// Mitsubishi GX Works2 project: SPMDanNhanV1   PLC: FX3G

// global labels: Global1
VAR_GLOBAL
  SIGNAL_JAR AT X000 : BOOL;
  SIGNAL_LABEL AT X001 : BOOL;
  EMERG AT X007 : BOOL;
  LABEL_PLS AT Y000 : BOOL;
  LABEL_DIR AT Y003 : BOOL;
  PushManLabel_F AT M200 : BOOL;
  PushManLabel_R AT M201 : BOOL;
  PushManGird_F AT M202 : BOOL;
  PushManGird_R AT M203 : BOOL;
  PushManRulo_F AT M204 : BOOL;
  PushManRulo_R AT M205 : BOOL;
  ModeAuto AT M206 : BOOL;
  Alarm AT M207 : BOOL;
  Operation AT M208 : BOOL;
  Speed_Label AT D200 : DINT;
  Length_Label AT D202 : DINT;
  Speed_Stamp AT D204 : DINT;
  Length_Stamp AT D206 : DINT;
  Round_Gird AT D208 : DINT;
  Round_Rulo AT D210 : DINT;
  Reset AT M209 : BOOL;
  Restore AT M210 : BOOL;
  FullStep_Label AT D212 : DINT;
  CommandLabel1 : BOOL;
  CommandLabel2 : BOOL;
  LABEL_ENB AT Y004 : BOOL;
  GIRD_PLS AT Y001 : BOOL;
  RULO_PLS AT Y002 : BOOL;
  RULO_ENB AT Y006 : BOOL;
  GIRD_ENB AT Y005 : BOOL;
  FinishPLS_Label AT M8340 : BOOL;
  Interrupt_GirdPLS AT M8350 : BOOL;
  Interrupt_RuloPLS AT M8360 : BOOL;
  PRINT_ENB AT Y007 : BOOL;
  RstCountStamp AT M211 : BOOL;
  Offset_Stamp AT D214 : DINT;
  CommandLabel : BOOL;
  Counter_Stamped AT D240 : DWORD;
  Time_Label AT D250 : DWORD;
  Counter_Label AT D8140 : DWORD;
  RatioDriver_Stamp : DINT;
END_VAR

// task Task_01 (event TRUE, interval 0, priority 31): POU_01
// task InterruptX000 (event I000, interval 0, priority 31): JAR
// task InterruptX001 (event I101, interval 0, priority 31): LABEL

PROGRAM POU_01
VAR
  Servo1_Label : Servo;
  ManualF_Label : BOOL;
  Servo2_Label : Servo;
  Restore_Q : BOOL;
  Freq_Label : DINT;
  Range_Label : DINT;
  Timer1_Label : TON_10;
  TimerPrint : TON_10;
  Timer_Restore : TON_10;
  Freq_Stamp : DINT;
  Range_Stamp : DINT;
  ManualR_Label : BOOL;
  Com1_Label : BOOL;
  Com2_Label : BOOL;
  TimerENB_Label : TON_10;
  TimerENB_Q : BOOL;
  TimerPrint_Q : BOOL;
END_VAR
EI( TRUE );
(* Khai bao vong quay va quang duong *)
DINCP ( SIGNAL_LABEL , Counter_Stamped );
SET( SIGNAL_LABEL AND SIGNAL_JAR, Alarm);
SET( LDP( TRUE, NOT SIGNAL_LABEL), PRINT_ENB);
TimerPrint( IN := PRINT_ENB, PT := T#100ms, Q := TimerPrint_Q);
RST( LDP( TRUE, TimerPrint_Q), PRINT_ENB);

Timer1_Label( IN := CommandLabel, PT := DWORD_TO_TIME( Time_Label), Q := Com1_Label );
SET( LDP( TRUE, Com1_Label), CommandLabel1);
RST( LDP( TRUE, Com1_Label), CommandLabel);

SET( LDF( TRUE, CommandLabel1), CommandLabel2);
DMOV(TRUE, Counter_Label, Round_Gird);

DMOV( NOT ModeAuto, 100*FullStep_Label, Freq_Label);
DMOV( ManualF_Label OR ManualR_Label, 20, Range_Label);

DMOV( ModeAuto, Speed_Label*FullStep_Label, Freq_Label);
DMOV( ModeAuto, Speed_stamp*FullStep_Label, Freq_Stamp);
DMOV( TRUE, Length_Label*RatioDriver_Stamp, Range_Label);
DMOV( TRUE, (Length_Label+Offset_Stamp)*RatioDriver_Stamp, Range_Stamp);

Servo1_Label( SetAutoMan := ModeAuto, 
							PushManF := ManualF_Label, PushManR := ManualR_Label,
							LimitInput := TRUE, LimitOutput := FinishPLS_Label, 
							Speed := Freq_Label, Range := Range_Label,
							SetAutoRunF := CommandLabel1, 
							OutputPLS := LABEL_PLS, OutputDIR := LABEL_DIR );

Servo2_Label( SetAutoMan := ModeAuto,
							LimitInput := TRUE, LimitOutput := FinishPLS_Label, 
							Speed := Freq_Stamp, Range := Range_Stamp,
							SetAutoRunF := CommandLabel2, OutputPLS := LABEL_PLS );

TimerENB_Label( IN := NOT FinishPLS_Label, PT := T#500ms, Q := TimerENB_Q);
LABEL_ENB := TimerENB_Q; 

Timer_Restore( IN := Restore, PT := T#5s, Q := Restore_Q );
IF Restore_Q THEN
	Speed_Label := 350;
	Speed_Stamp := 350;
	Length_Label := 70;
	FullStep_Label := 8;
	Time_Label := 300;
	Offset_Stamp := 0;
END_IF;

IF RstCountStamp THEN
	Counter_Stamped := 0;
END_IF;

IF Reset THEN
	Alarm := FALSE;
	Com1_Label := FALSE;
	CommandLabel1 := FALSE;
	CommandLabel2 := FALSE;
END_IF;

(*NGUYEN LY: Kich chay Step 2 lan
Lan 1: khi phat hien co chai, delay Time_Label ms -> run toi khi SIGNAL_LABEL = ON thi dung
Lan 2: khi SIGNAL_LABEL = ON chay lai Step het quang duong thi dung.
Ly do: de danh Command1 doi chai tiep theo
do duong kinh ong bang encoder: khi ong di qua cam bien lay xung canh len - dem encoder counter,
khi ong qua het lay xung canh xuong doc encoder counter
*)
(*
MUL_E( TRUE , Speed_Label , 166.67 , Speed_Stamp );
REAL_TO_DINT_E( TRUE , Speed_Stamp , Speed_Label );

*)
END_PROGRAM

FUNCTION_BLOCK Servo
VAR_INPUT
  SetAutoMan : BOOL;
  Speed : DINT;
  Range : DINT;
END_VAR
VAR_IN_OUT
  SetAutoRunF : BOOL;
  SetAutoRunR : BOOL;
END_VAR
VAR_OUTPUT
  OutputPLS : BOOL;
  OutputDIR : BOOL;
END_VAR
VAR
  RelayPLS : BOOL;
  RelayDIR : BOOL;
END_VAR
VAR_IN_OUT
  PushManF : BOOL;
  PushManR : BOOL;
END_VAR
VAR_INPUT
  LimitOutput : BOOL;
  LimitInput : BOOL;
END_VAR
(* Set mode Auto/Man *)
IF  SetAutoMan THEN
	RelayDIR := SetAutoRunR;
	RelayPLS := SetAutoRunF OR SetAutoRunR;
ELSE
	RelayDIR := PushManR;
	RelayPLS := PushManF OR PushManR;
END_IF;

OutputDIR := RelayDIR ;

DPLSY( RelayPLS AND LimitInput, Speed, Range , OutputPLS );

(* Reset control signal *)
RST( LDF( TRUE, LimitOutput ) , SetAutoRunF );
RST( LDF( TRUE, LimitOutput) , SetAutoRunR );
RST( LDF( TRUE, LimitOutput ) , PushManF );
RST( LDF( TRUE, LimitOutput) , PushManR );
END_FUNCTION_BLOCK

PROGRAM JAR
SET( TRUE, CommandLabel);
END_PROGRAM

PROGRAM LABEL
RST( TRUE, CommandLabel1);
RST( TRUE, Counter_Label);
END_PROGRAM
